KUKA KRL program: Lequn_MRP_TopLeft_XY_no_rsi.src, Lequn_MRP_TopLeft_XY_no_rsi.dat

--- Lequn_MRP_TopLeft_XY_no_rsi.src ---
&ACCESS RVO
&REL 193
&PARAM DISKPATH = KRC:\R1\Program\Lequn
DEF Lequn_MRP_TopLeft_XY_no_rsi( )

   DECL E6POS LayerStartPt
   DECL E6POS LayerStartPt2
   DECL E6POS LayerStartPt3
   DECL E6POS LayerStartPt4
   DECL E6POS XP2
   DECL E6POS XP3
   DECL E6POS XP4
   DECL REAL stepover
   DECL REAL xLength
   DECL REAL yWidth
   DECL REAL layerHt
   DECL INT YSTEP
   DECL INT YSTEP_MAX
   DECL INT XSTEP
   DECL INT XSTEP_MAX
   DECL INT nLayers ;  the total number of layers
   DECL INT layer ; the current layer number
   DECL REAL power
   DECL INT countOdd;
   DECL INT countEven;
   DECL INT oddEven;


   GLOBAL INTERRUPT DECL 3 WHEN $STOPMESS==TRUE DO IR_STOPM ( )
   INTERRUPT ON 3
   BAS (#INITMOV,0 )

   ptp $POS_ACT

   ;FOLD LIN P1 Vel=0.02 m/s CPDAT1 Tool[1]:LASER Base[0] ;%{PE}
      ;FOLD Parameters ;%{h}
         ;Params IlfProvider=kukaroboter.basistech.inlineforms.movement.old; Kuka.IsGlobalPoint=False; Kuka.PointName=P1; Kuka.BlendingEnabled=False; Kuka.MoveDataName=CPDAT1; Kuka.VelocityPath=0.02; Kuka.CurrentCDSetIndex=0; Kuka.MovementParameterFieldEnabled=True; IlfCommand=LIN
      ;ENDFOLD

      $BWDSTART = FALSE
      LDAT_ACT = LCPDAT1
      FDAT_ACT = FP1
      BAS(#CP_PARAMS, 0.02)
      SET_CD_PARAMS (0)
      LIN XP1
   ;ENDFOLD

   ;--------------Process variables-----------------
   stepover = 1.0 ;mm
   xLength = 90.0 ;mm
   yWidth = 20.0 ;mm
   layerHt = 0.85 ;mm
   nLayers = 10

   $VEL.CP=0.022 ; feed rate in m/s
   $APO.CDIS = 0.24 ; mm ; equivalent to Zone data in ABB (Z0)
   $ANOUT[1]= 0.205 ;0.180 ; laser power in voltage
   ;$ANOUT[2]=0.2125 ; wire feed rate in voltage
   ;-------------------------------------------------

   LIN XP1

   $OUT[15]=TRUE ; Wire touch signal bypass

   LaserOn_Ext() ; on laser
   countOdd = 1
   countEven = 1
   For layer = 1 TO nLayers STEP 1
      IF(layer/2) <>(layer/2.0) THEN
         ;odd layer

         ; move to start point
         LayerStartPt = XP1
         LayerStartPt.Z = XP1.Z + layerHt * (layer - 1)
         LayerStartPt.Y = LayerStartPt.Y - stepover*2

         ;layer1 or layer3

         ;; find out if it a layer 1 or layer
         IF(countOdd/2) <>(countOdd/2.0)THEN
            oddEven = 1
            YSTEP_MAX = yWidth / stepover
            FOR YSTEP = 0 TO YSTEP_MAX
               ;; layer 1
               IF(oddEven/2) <>(oddEven/2.0)THEN

                  LayerStartPt.Y = LayerStartPt.Y + stepover*2

                  XP2 = LayerStartPt
                  XP2.X = XP2.X + xLength
                  LIN LayerStartPt

                  LaserStart_Ext()
                  LIN XP2

                  ;WAIT SEC 0.2
                  LaserEnd_Ext()

                  oddEven = oddEven+1
               ELSE
                  XP3 = XP2

                  XP3.Y = XP3.Y + stepover
                  LIN XP3
                  XP4 = XP3
                  XP4.X = XP4.X - xLength

                  LaserStart_Ext()
                  LIN XP4

                  ;WAIT SEC 0.2
                  LaserEnd_Ext()

                  oddEven = oddEven +1
               ENDIF

            ENDFOR

            countOdd = countOdd +1

         ELSE
            oddEven =1
            YSTEP_MAX = yWidth / stepover
            LayerStartPt3 = XP1
            LayerStartPt3.Z = LayerStartPt3.Z + layerHt * (layer - 1)
            LayerStartPt3.x = LayerStartPt3.X + xLength
            LayerStartPt3.y = LayerStartPt3.y + yWidth
            ;; move to layer 3 start point bottom right
            LIN LayerStartPt3
            WAIT SEC 1.0
            LayerStartPt3.y = LayerStartPt3.y + stepover * 2

            FOR YSTEP = 0 TO YSTEP_MAX
               ;; layer 3
               IF(oddEven/2) <>(oddEven/2.0)THEN

                  LayerStartPt3.y = LayerStartPt3.y - stepover * 2

                  LIN LayerStartPt3
                  XP2 = LayerStartPt3
                  XP2.X = XP2.X - xLength

                  LaserStart_Ext()
                  LIN XP2

                  LaserEnd_Ext()
                  oddEven = oddEven + 1
               ELSE

                  XP3 = XP2
                  XP3.Y = XP3.Y - stepover
                  LIN XP3
                  XP4 = XP3
                  XP4.X = XP4.X + xLength

                  LaserStart_Ext()
                  LIN XP4
                  ;WireFeederOff()
                  ;WAIT SEC 0.2
                  LaserEnd_Ext()

                  oddEven = oddEven + 1
               ENDIF

            ENDFOR
            countOdd = countOdd +1
         ENDIF

         LaserEnd_Ext()

      ELSE

         ;even layer
         ;layer 2
         IF(countEven/2) <>(countEven/2.0)THEN
            oddEven = 1
            LayerStartPt2 = XP1
            LayerStartPt2.Z = XP1.Z + layerHt * (layer - 1)
            LayerStartPt2.X = LayerStartPt2.X + xLength

            LIN LayerStartPt2
            WAIT SEC 1.0

            LayerStartPt2.X = LayerStartPt2.X + stepover*2
            XSTEP_MAX = xLength / stepover

            FOR XSTEP = 1 to XSTEP_MAX
               ;;LAYER 2
               IF(oddEven/2) <>(oddEven/2.0)THEN
                  LayerStartPt2.X = LayerStartPt2.X - stepover*2
                  XP2 = LayerStartPt2

                  LIN LayerStartPt2

                  LaserStart_Ext()
                  XP2.Y = XP2.Y + yWidth
                  LIN XP2
                  LaserEnd_Ext()

                  oddEven = oddEven + 1
               ELSE

                  XP3 = XP2
                  XP3.X = XP3.X - stepover
                  LIN XP3
                  XP4 = XP3
                  XP4.Y = XP4.Y - yWidth

                  LaserStart_Ext()
                  LIN XP4
                  LaserEnd_Ext()

                  oddEven = oddEven + 1
               ENDIF
            ENDFOR
            countEven = countEven +1
         ELSE
            ;; even layer layer 4
            oddEven = 1
            LayerStartPt4 = XP1
            LayerStartPt4.z = XP1.Z + layerHt * (layer - 1)
            XSTEP_MAX = xLength / stepover

            LayerStartPt4.y = LayerStartPt4.y + yWidth

            LIN LayerStartPt4
            WAIT SEC 1.0
            LayerStartPt4.X = LayerStartPt4.X - stepover*2

            FOR XSTEP = 1 to XSTEP_MAX
               ;;LAYER 4
               IF(oddEven/2) <>(oddEven/2.0)THEN
                  LayerStartPt4.X = LayerStartPt4.X + stepover*2
                  XP2 = LayerStartPt4

                  LIN LayerStartPt4
                  XP2.Y = XP2.Y - yWidth

                  LaserStart_Ext()
                  LIN XP2
                  LaserEnd_Ext()

                  oddEven = oddEven + 1

               ELSE

                  XP3 = XP2
                  XP3.X = XP3.X + stepover
                  LIN XP3
                  XP4 = XP3
                  XP4.Y = XP4.Y + yWidth

                  LaserStart_Ext()
                  LIN XP4
                  LaserEnd_Ext()
                  oddEven = oddEven + 1
               ENDIF

            ENDFOR
            countEven = countEven +1
         ENDIF
         LaserEnd_Ext()

      ENDIF
   ENDFOR
   LaserOff_Ext()

   $OUT[15]=FALSE ; Deactivate wire touch signal bypass

END

--- Lequn_MRP_TopLeft_XY_no_rsi.dat ---
&ACCESS RVO
&REL 193
&PARAM DISKPATH = KRC:\R1\Program\Lequn
DEFDAT  Lequn_MRP_TopLeft_XY_no_rsi
;FOLD EXTERNAL DECLARATIONS;%{PE}%MKUKATPBASIS,%CEXT,%VCOMMON,%P
;FOLD BASISTECH EXT;%{PE}%MKUKATPBASIS,%CEXT,%VEXT,%P
EXT  BAS (BAS_COMMAND  :IN,REAL  :IN )
DECL INT SUCCESS
;ENDFOLD (BASISTECH EXT)
;FOLD USER EXT;%{E}%MKUKATPUSER,%CEXT,%VEXT,%P
;Make your modifications here

;ENDFOLD (USER EXT)
;ENDFOLD (EXTERNAL DECLARATIONS)
DECL E6POS XP1={X 3017.01807,Y -1705.93262,Z 919.358521,A -90.1117935,B -0.497298241,C 177.995636,S 22,T 51,E1 -1324.94983,E2 0.00722303381,E3 -0.715565,E4 0.0,E5 0.0,E6 0.0}
DECL FDAT FP1={TOOL_NO 1,BASE_NO 0,IPO_FRAME #BASE,POINT2[] " "}
DECL LDAT LCPDAT1={VEL 0.0200000,ACC 100.000,APO_DIST 500.000,APO_FAC 50.0000,AXIS_VEL 100.000,AXIS_ACC 100.000,ORI_TYP #VAR,CIRC_TYP #BASE,JERK_FAC 50.0000,GEAR_JERK 100.000,EXAX_IGN 0}
DECL MODULEPARAM_T LAST_TP_PARAMS={PARAMS[] "Kuka.PointName=P1; Kuka.FrameData.base_no=0; Kuka.FrameData.tool_no=1; Kuka.FrameData.ipo_frame=#BASE; Kuka.isglobalpoint=False; Kuka.MoveDataName=CPDAT1; Kuka.MovementData.apo_fac=50; Kuka.MovementData.apo_dist=500; Kuka.MovementData.axis_acc=100; Kuka.MovementData.axis_vel=100; Kuka.MovementData.circ_typ=#BASE; Kuka.MovementData.jerk_fac=50; Kuka.MovementData.ori_typ=#VAR; Kuka.MovementData.vel=0.02; Kuka.MovementData.acc=100; Kuka.MovementData.exax_ign=0; Kuka.VelocityPath=0.02; Kuka.BlendingEnabled=False; Kuka.CurrentCDSetIndex=0; SyncLabel=AutoSync; Kuka.FrameData.point2=      "}
DECL E6POS XP5={X 1267.51770,Y -1547.66406,Z 1189.19409,A -89.9841156,B -0.616697371,C 178.079834,S 22,T 51,E1 -1150.03894,E2 0.00427939091,E3 -1.87918558E-05,E4 0.0,E5 0.0,E6 0.0}
ENDDAT
